// Implicitly generated code : DO NOT EDIT
FUNCTION CheckLRangeUnsigned : ULINT
VAR_INPUT
    value, lower, upper: ULINT;
END_VAR

// Implicitly generated code : Only an Implementation suggestion
{noflow}
IF (value < lower) THEN
    CheckLRangeUnsigned := lower;
ELSIF(value > upper) THEN
    CheckLRangeUnsigned := upper;
ELSE
    CheckLRangeUnsigned := value;
END_IF
{flow}

END_FUNCTION

(* stored: Version 1.1.0.1, ProductVersion 3.1.4024.6
   POU CheckLRangeUnsigned: Id {b292ab2e-8e75-41b2-a9d3-2a4bb6be970c}, SpecialFunc CheckLRangeUnsigned *)
